// TIA Portal V18 export
DATA_BLOCK "CMMS_Z1_Movement_DB"   // DB76
VERSION : 0.1
// stored: AutoNumber true, DBAccessibleFromOPCUA true, InstanceOfName CMMS_Z1_Movement, InstanceOfType FB
"CMMS_Z1_Movement"
   // VAR
   //    FML_REF { S7_SetPoint := 'True'} : "DT_FML_REF";
   // END_VAR
BEGIN
END_DATA_BLOCK
